FUNCTION_BLOCK fbSlowPullAxisCtrl
VAR_INPUT

	bPosStart : BOOL;
	bHomingRdy : BOOL;
	wTargetPosNum : WORD;
	lrDownVelo : LREAL;
	lrDownAcc : LREAL;
	lrDownDcc : LREAL;
	lrDownVelo2 : LREAL;
	lrDownAcc2 : LREAL;
	lrDownDcc2 : LREAL;
	lrUpVelo : LREAL;
	lrUpAcc : LREAL;
	lrUpDcc : LREAL;
	lrUpVelo2 : LREAL;
	lrUpAcc2 : LREAL;
	lrUpDcc2: LREAL;
	lrCurrentServoPos : LREAL;
	lrDownPos : LREAL;
	lrUpPos : LREAL;
	lrUpAgitationPos : LREAL;
	lrDownAgitationPos : LREAL;

END_VAR

VAR_IN_OUT

	ArmLifter : axis_ref;
END_VAR

VAR_OUTPUT

	AxisStopEn : BOOL;

END_VAR
VAR

	Halt1: MC_Halt;
	Stoptimer: TON;
	AxisStopbit: BOOL;
	TimerMove: TON;
	BlockStartBit: BOOL;
	Move1: BOOL;
	Move2: BOOL;
	Move3: BOOL;
	Move4: BOOL;
	Move5: BOOL;
	Move6: BOOL;
	Move7: BOOL;
	Move8: BOOL;
	Move9: BOOL;
	Move10: BOOL;
	Move11: BOOL;
	Move12: BOOL;
	Move13: BOOL;
	Move14: BOOL;
	Move15: BOOL;
	Move16: BOOL;
	Move17: BOOL;
	Move18: BOOL;
	Move19: BOOL;
	Move20: BOOL;
	Halt2: MC_Halt;
	ArmMoveTostation2: MC_MoveAbsolute;
	ArmMoveTostation: MC_MoveAbsolute;
	PosSV: LREAL;
	AccSv: LREAL;
	DccSv: LREAL;
	VeloSv: LREAL;
	Arm2ndSpeedEnable: BOOL;

END_VAR
VAR // added by the converter: edge detectors and wires of the graphical bodies
    _w1, _w2, _w3, _w4, _w5, _w6, _w7, _w8, _w9, _w10, _w11, _w12, _w13, _w14, _w15, _w16 : LREAL;
END_VAR

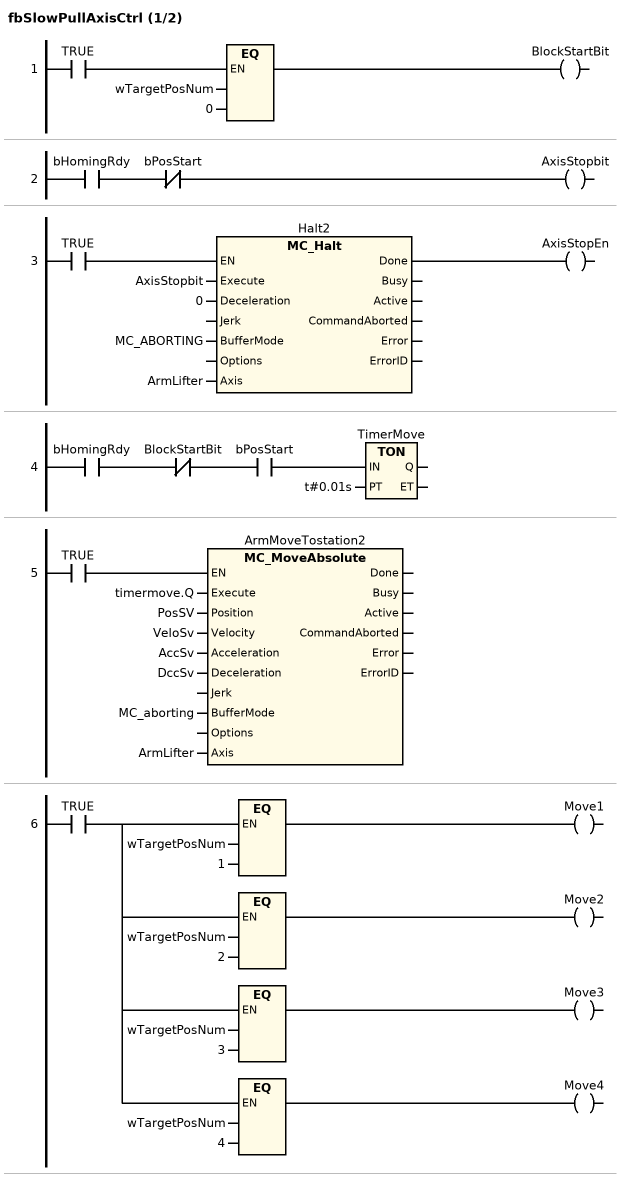
// NETWORK 1
BlockStartBit := wTargetPosNum = 0;

// NETWORK 2
AxisStopbit := bHomingRdy AND NOT bPosStart;

// NETWORK 3
Halt2(Execute := AxisStopbit, Deceleration := 0, BufferMode := MC_ABORTING, Axis := ArmLifter); // MC_Halt
AxisStopEn := Halt2.Done;

// NETWORK 4
TimerMove(IN := bHomingRdy AND NOT BlockStartBit AND bPosStart, PT := t#0.01s); // TON

// NETWORK 5
ArmMoveTostation2(
    Execute := timermove.Q,
    Position := PosSV,
    Velocity := VeloSv,
    Acceleration := AccSv,
    Deceleration := DccSv,
    BufferMode := MC_aborting,
    Axis := ArmLifter); // MC_MoveAbsolute

// NETWORK 6
Move1 := wTargetPosNum = 1;
Move2 := wTargetPosNum = 2;
Move3 := wTargetPosNum = 3;
Move4 := wTargetPosNum = 4;

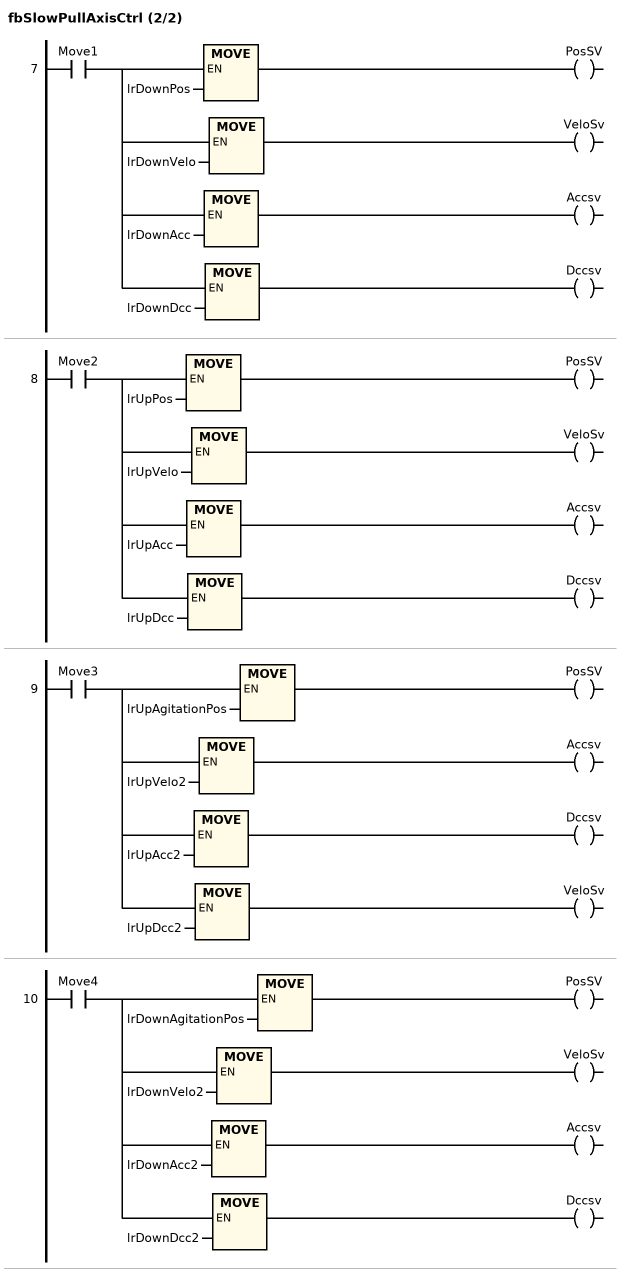
// NETWORK 7
IF Move1 THEN _w1 := lrDownPos; END_IF
PosSV := _w1;
IF Move1 THEN _w2 := lrDownVelo; END_IF
VeloSv := _w2;
IF Move1 THEN _w3 := lrDownAcc; END_IF
Accsv := _w3;
IF Move1 THEN _w4 := lrDownDcc; END_IF
Dccsv := _w4;

// NETWORK 8
IF Move2 THEN _w5 := lrUpPos; END_IF
PosSV := _w5;
IF Move2 THEN _w6 := lrUpVelo; END_IF
VeloSv := _w6;
IF Move2 THEN _w7 := lrUpAcc; END_IF
Accsv := _w7;
IF Move2 THEN _w8 := lrUpDcc; END_IF
Dccsv := _w8;

// NETWORK 9
IF Move3 THEN _w9 := lrUpAgitationPos; END_IF
PosSV := _w9;
IF Move3 THEN _w10 := lrUpVelo2; END_IF
Accsv := _w10;
IF Move3 THEN _w11 := lrUpAcc2; END_IF
Dccsv := _w11;
IF Move3 THEN _w12 := lrUpDcc2; END_IF
VeloSv := _w12;

// NETWORK 10
IF Move4 THEN _w13 := lrDownAgitationPos; END_IF
PosSV := _w13;
IF Move4 THEN _w14 := lrDownVelo2; END_IF
VeloSv := _w14;
IF Move4 THEN _w15 := lrDownAcc2; END_IF
Accsv := _w15;
IF Move4 THEN _w16 := lrDownDcc2; END_IF
Dccsv := _w16;

END_FUNCTION_BLOCK

(* stored: Version 1.1.0.1, ProductVersion 3.1.4024.12
   POU fbSlowPullAxisCtrl: Id {3170d5be-8991-450c-a2ac-3b56459765a3}, SpecialFunc None *)
